TYPE Millisecond : LREAL; END_TYPE

(* stored: Version 1.1.0.1
   DUT Millisecond: Id {02e4c6ff-f486-4de8-9a70-ddf04d675dc3} *)
